(* IEC 61131-3 sources: volt/packages/volt-lsp-iec/test-corpus/awa-palletizer/Device/Plc Logic/Application/Library Manager/SysSemProcess, 5 files *)

(* ---- GLOBAL_CONSTANTS.gvl ---- *)
VAR_GLOBAL
	SYSSEMPROCESS_INVALID_HANDLE : UDINT := 16#FFFFFFFF;
END_VAR

(* ---- SYSSEMPROCESSCREATE.pou ---- *)
FUNCTION SYSSEMPROCESSCREATE : RTS_IEC_HANDLE
VAR_INPUT
	PSZNAME : REFERENCE TO STRING;
	PRESULT : POINTER TO RTS_IEC_RESULT;
END_VAR
END_FUNCTION

(* ---- SYSSEMPROCESSDELETE.pou ---- *)
FUNCTION SYSSEMPROCESSDELETE : RTS_IEC_RESULT
VAR_INPUT
	HSEM : RTS_IEC_HANDLE;
END_VAR
END_FUNCTION

(* ---- SYSSEMPROCESSENTER.pou ---- *)
FUNCTION SYSSEMPROCESSENTER : RTS_IEC_RESULT
VAR_INPUT
	HSEM : RTS_IEC_HANDLE;
	ULTIMEOUT : UDINT;
END_VAR
END_FUNCTION

(* ---- SYSSEMPROCESSLEAVE.pou ---- *)
FUNCTION SYSSEMPROCESSLEAVE : RTS_IEC_RESULT
VAR_INPUT
	HSEM : RTS_IEC_HANDLE;
END_VAR
END_FUNCTION
